{attribute addProperty BoxType "IODEVICETYPE_ETHERCATPROT"}
{attribute addProperty Id "Beckhoff_AT1xxxBeckhoff_AT1xxx_7510A45A461125764Beckhoff_ATH2xxxBeckhoff_ATH2xxx_159CB27D6890861.25SyncUnitsSyncUnits_CAB22D3B19524.375InputsInputs_C75D3FEC1280160OutputsOutputs_47D1E803848106InfoDataInfoData_E9F65A829612"}
{attribute addProperty CRC "2204574006"}
{attribute addProperty SizeInBites "55421"}
{attribute addProperty SizeInBytes "6927.625"}
TYPE EtherCAT_Master_ATxxxx_83672136 :
STRUCT
	{attribute addProperty Name "Beckhoff_AT1xxx"}
	Beckhoff_AT1xxx : Beckhoff_AT1xxx_7510A45A;
	{attribute addProperty Name "Beckhoff_ATH2xxx"}
	Beckhoff_ATH2xxx : Beckhoff_ATH2xxx_159CB27D;
	{attribute addProperty Name "SyncUnits"}
	SyncUnits : SyncUnits_CAB22D3B;
	{attribute addProperty Name "Inputs"}
	Inputs : Inputs_C75D3FEC;
	{attribute addProperty Name "Outputs"}
	Outputs : Outputs_47D1E803;
	{attribute addProperty Name "InfoData"}
	InfoData : InfoData_E9F65A82;
END_STRUCT
END_TYPE

(* stored: Version 1.2.0.0, ProductVersion 3.1.4024.9
   DUT EtherCAT_Master_ATxxxx_83672136: Id {6e76b621-7d91-4869-bf98-8b3de0db35de} *)
